{attribute 'linkalways'} 
{attribute 'no_explicit_call' := 'This FB is a CLASS and must be accessed using methods or properties'}
{attribute 'enable_dynamic_creation'}
FUNCTION_BLOCK FINAL MIN_USINT EXTENDS Node
VAR
	in1 : _USINT(0);
	in2 : _USINT(0);
	out : _USINT(0);
END_VAR

METHOD PUBLIC Clone : I_Node
VAR
	pNode : POINTER TO MIN_USINT;
END_VAR
pNode := __NEW(MIN_USINT);
Clone := pNode^;
END_METHOD

METHOD FB_init : BOOL
VAR_INPUT
	bInitRetains : BOOL; // if TRUE, the retain variables are initialized (warm start / cold start)
	bInCopyCode : BOOL;  // if TRUE, the instance afterwards gets moved into the copy code (online change)
END_VAR
AddInput('in1',THIS^.in1);
AddInput('in2',THIS^.in2);
AddOutput('out', THIS^.out);
END_METHOD

METHOD PROTECTED OnExecute
VAR
END_VAR
out.Value := MIN(in1.Value, in2.Value);
END_METHOD

END_FUNCTION_BLOCK

(* stored: Version 1.1.0.1, ProductVersion 3.1.4024.15
   POU MIN_USINT: Id {a8dcfb9f-44d1-4a16-a26f-be61b6d8c863}, SpecialFunc None
   Folder Constructor: Id {4e039580-1ee4-410e-893f-42e55ae48ce9}
   Method Clone: Id {86db378d-c164-4b2e-8f2a-155e363fafb9}
   Method FB_init: Id {6f6bacac-6caf-4a0a-a3f7-300c0a71440f}
   Method OnExecute: Id {3a026dd1-9812-4c1d-a82f-864a921b1e06} *)
